% RSLogix 500 project AND_Program.RSS, saved by version 8.30.00.16 %
PROJECT "AND'"    % processor: Bul.1763 MicroLogix 1100 Series B %

PROGRAM FILES
  LAD 2   2 rungs

DATA FILES
  O0 OUTPUT  4 elements
  I1 INPUT  6 elements
  S2 STATUS  66 elements
  B3 BINARY  1 elements
  T4 TIMER  1 elements
  C5 COUNTER  1 elements
  R6 CONTROL  1 elements
  N7 INTEGER  1 elements
  F8 FLOAT  1 elements

LADDER 2
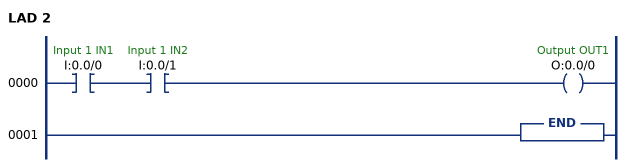
% Rung: 0 %
SOR XIC I:0.0/0 XIC I:0.0/1 OTE O:0.0/0 EOR
%   I:0.0/0  IN1  "Input 1" %
%   I:0.0/1  IN2  "Input 1" %
%   O:0.0/0  OUT1  "Output" %
% Rung: 1 %
SOR END EOR
